      sx_ReqInProgress380 { ExternalAccessible := 'False'; ExternalVisible := 'False'; ExternalWritable := 'False'} : Bool;   // Request for 380 is in progress
      sx_ReqInProgress390 { ExternalAccessible := 'False'; ExternalVisible := 'False'; ExternalWritable := 'False'} : Bool;   // Request for 390 is in progress
      sx_ActiveRequest680 { ExternalAccessible := 'False'; ExternalVisible := 'False'; ExternalWritable := 'False'} : Bool;   // Request for 680 is active
      sx_ActiveRequest690 { ExternalAccessible := 'False'; ExternalVisible := 'False'; ExternalWritable := 'False'} : Bool;   // Request for 690 is active
      sx_ReqInProgress680 { ExternalAccessible := 'False'; ExternalVisible := 'False'; ExternalWritable := 'False'} : Bool;   // Request for 680 is in progress
      sx_ReqInProgress690 { ExternalAccessible := 'False'; ExternalVisible := 'False'; ExternalWritable := 'False'} : Bool;   // Request for 690 is in progress
      sx_TransferOut380 { ExternalAccessible := 'False'; ExternalVisible := 'False'; ExternalWritable := 'False'} : Bool;   // Transfer out from 380 is active
      sx_TransferOut390 { ExternalAccessible := 'False'; ExternalVisible := 'False'; ExternalWritable := 'False'} : Bool;   // Transfer out from 390 is active
      sx_TransferOut680 { ExternalAccessible := 'False'; ExternalVisible := 'False'; ExternalWritable := 'False'} : Bool;   // Transfer out from 680 is active
      sx_TransferOut690 { ExternalAccessible := 'False'; ExternalVisible := 'False'; ExternalWritable := 'False'} : Bool;   // Transfer out from 690 is active
      sx_DirectionChange380 { ExternalAccessible := 'False'; ExternalVisible := 'False'; ExternalWritable := 'False'} : Bool;   // Direction of conveyor 380
      sx_DirectionChange390 { ExternalAccessible := 'False'; ExternalVisible := 'False'; ExternalWritable := 'False'} : Bool;   // Direction of conveyor 390
      sx_DirectionChange680 { ExternalAccessible := 'False'; ExternalVisible := 'False'; ExternalWritable := 'False'} : Bool;   // Direction of conveyor 680
      sx_DirectionChange690 { ExternalAccessible := 'False'; ExternalVisible := 'False'; ExternalWritable := 'False'} : Bool;   // Direction of conveyor 690
      sx_Hold230 { ExternalAccessible := 'False'; ExternalVisible := 'False'; ExternalWritable := 'False'} : Bool;
      sx_Hold530 { ExternalAccessible := 'False'; ExternalVisible := 'False'; ExternalWritable := 'False'} : Bool;
      sx_ClearRightStation { ExternalAccessible := 'False'; ExternalVisible := 'False'; ExternalWritable := 'False'} : Bool;   // Command to clear right station
      sx_ClearLeftStation { ExternalAccessible := 'False'; ExternalVisible := 'False'; ExternalWritable := 'False'} : Bool;   // Command to clear left station
   END_VAR

   VAR_TEMP
      tUDT_dummyHandshake : "UDT_ConveyorHandshake";   // Dummy handshake structure
      tUDT_DummyBladeStop : "UDT_ValveInterface";
      ts_Barcode110 : String;
      ts_Barcode330 : String;
      ts_Barcode630 : String;
      tw_dummy : Word;
      ti_dummy : Int;   // Dummy int
      tx_dummy : Bool;   // Dummy bool
   END_VAR


BEGIN
	(*
	----------------------------------------------------------------------------------------

	Version history:
	Date        | Version   | Author        | Remark
	----------------------------------------------------------------------------------------
	23/02/2024  | 0.1       | R. Pieczonka  | Initial version
	26/02/2024  | 0.2       | S. Nieswiec   | Updated to new library blocks, added HardwareOk input
	27/02/2024  | 0.3       | S. Nieswiec   | Mapped  safetyOk, 24vOk, 400vOk from inputs to function blocks, added VFDs in place of conveylinx at conveyors 260,310,560,610
	18/03/2024  | 0.4       | S. Nieswiec   | Adjusted comments and variable names
	15/04/2024  | 0.5       | S. Nieswiec   | Added ConveyLinx Controllers
	10/05/2024  | 0.6       | R. Pieczonka  | Added new MCO and clearing sequence. Changes in station operation sequence.
	04/06/2024  | 0.7       | S. Nieswiec   | Partially added scanners
	11/06/2024  | 0.8       | S. Nieswiec   | New RAT, MCO and Displacement FB + added datalogic scanner
	14/06/2024  | 0.9       | S. Nieswiec   | New RAT, MCO and Displacement FB + added datalogic scanner
	*)
	(*
	----------------------------------------------------------------------------------------

	Notes:
	Date        | Version   | Author        | Notes
	----------------------------------------------------------------------------------------
	25/06/2024  | 0.9       | I.Bou Ajram   | Barcode scanners and the use of external DBs directly needs tidying up. request update


	*)

	REGION Middle line - Infeed
	    (*
	    REGION 010

	        REGION Displacement

	            #sFB_Displacement010(#sUDT_Interface_010);

	        END_REGION

	        REGION Conveyor
	            #sFB_Conveyor_010(iUDT_ConveyorConfiguration := #iUDT_Configuration."010".Conveyor,
	                              idi_PECEoSDistance         := 0,
	                              idi_PECBoSDistance         := 0,
	                              ii_ExternalSpeed           := 0,
	                              ix_SafetyOk                := #ix_SafetyOk,
	                              ix_24vOk                   := #ix_24vOk,
	                              ix_400vOk                  := #ix_400vOk,
	                              ix_HardwareOk              := #ix_HardwareOk,
	                              ix_PECEoS                  := TRUE,
	                              ix_PECBoS                  := TRUE,
	                              ix_ExternalRequestHold     := false,
	                              qUDT_HMIStatus             => #iqUDT_WorkstationStatus."010".Conveyor,
	                              qUDT_Status                => #iqUDT_WorkstationCommonStatus."010",
	                              iqUDT_EquipmentControl     := #iqUDT_EquipmentControl,
	                              iqUDT_ConveyorCommand      := #iqUDT_WorkstationCommands."010",
	                              iqUDT_ConveyorInterface    := #sUDT_Interface_010,
	                              iqUDT_HandShakeUp          := #iqUDT_HandshakeUpstream010,
	                              iqUDT_HandShake            := #sUDT_Handshake_010,
	                              iqUDT_Statistics           := #iqUDT_WorkstationStatistics."010".Conveyor);
	        END_REGION

	        REGION MCO
	            #sFB_MCOConveyLinxAixController_010(iUDT_AixConfig          := #iUDT_Configuration."010".MCO,
	                                                iUDT_AixInputsModule    := #iUDT_MotorInput010,
	                                                ix_24vOk                := #ix_24vOk,
	                                                ix_SimulationModeActive := "DB_Memory".Simulation,
	                                                ii_MotorPositionId      := 1,
	                                                qUDT_HMIStatus          => #iqUDT_WorkstationStatus."010".MCO,
	                                                iqUDT_AixOutputsModule  := #qUDT_MotorOutput010,
	                                                iqUDT_ConveyorInterface := #sUDT_Interface_010,
	                                                iqUDT_MCOStatistics     := #iqUDT_WorkstationStatistics."010".MCO);
	        END_REGION
	    END_REGION


	    REGION 020

	        REGION Displacement

	            #sFB_Displacement020(#sUDT_Interface_020);

	        END_REGION

	        REGION EoS

	            #sFB_PEC_020(ix_PEC                   := #iUDT_MotorInput020.AllSensorPortInputs.LeftSensor,
	                         iUDT_PECConfiguration   := #iUDT_Configuration."020".PEC_Eos,
	                         qUDT_HMIStatus          => #iqUDT_WorkstationStatus."020".PEC_Eos,
	                         iqUDT_ConveyorInterface := #sUDT_Interface_020,
	                         iqUDT_PECStatistics     := #iqUDT_WorkstationStatistics."020".PEC_Eos);

	        END_REGION

	        REGION Conveyor
	            #sFB_Conveyor_020(iUDT_ConveyorConfiguration := #iUDT_Configuration."020".Conveyor,
	                              idi_PECEoSDistance         := #iUDT_Configuration."020".PEC_Eos.Distance,
	                              idi_PECBoSDistance         := 0,
	                              ii_ExternalSpeed           := 0,
	                              ix_SafetyOk                := #ix_SafetyOk,
	                              ix_24vOk                   := #ix_24vOk,
	                              ix_400vOk                  := #ix_400vOk,
	                              ix_HardwareOk              := #ix_HardwareOk,
	                              ix_PECEoS                  := #iqUDT_WorkstationStatus."020".PEC_Eos.PEC,
	                              ix_PECBoS                  := TRUE,
	                              ix_ExternalRequestHold     := false,
	                              qUDT_HMIStatus             => #iqUDT_WorkstationStatus."020".Conveyor,
	                              qUDT_Status                => #iqUDT_WorkstationCommonStatus."020",
	                              iqUDT_EquipmentControl     := #iqUDT_EquipmentControl,
	                              iqUDT_ConveyorCommand      := #iqUDT_WorkstationCommands."020",
	                              iqUDT_ConveyorInterface    := #sUDT_Interface_020,
	                              iqUDT_HandShakeUp          := #sUDT_Handshake_010,
	                              iqUDT_HandShake            := #sUDT_Handshake_020,
	                              iqUDT_Statistics           := #iqUDT_WorkstationStatistics."020".Conveyor);
	        END_REGION

	        REGION MCO
	            #sFB_MCOConveyLinxAixController_020(iUDT_AixConfig          := #iUDT_Configuration."020".MCO,
	                                                iUDT_AixInputsModule    := #iUDT_MotorInput020,
	                                                ix_24vOk                := #ix_24vOk,
	                                                ix_SimulationModeActive := "DB_Memory".Simulation,
	                                                ii_MotorPositionId      := 1,
	                                                qUDT_HMIStatus          => #iqUDT_WorkstationStatus."020".MCO,
	                                                iqUDT_AixOutputsModule  := #qUDT_MotorOutput020,
	                                                iqUDT_ConveyorInterface := #sUDT_Interface_020,
	                                                iqUDT_MCOStatistics     := #iqUDT_WorkstationStatistics."020".MCO);
	        END_REGION


	    END_REGION

	    REGION 030

	        REGION Displacement

	            #sFB_Displacement030(#sUDT_Interface_030);

	        END_REGION

	        REGION EoS

	            #sFB_PEC_030(ix_PEC                   := #iUDT_MotorInput030.AllSensorPortInputs.LeftSensor,
	                         iUDT_PECConfiguration   := #iUDT_Configuration."030".PEC_Eos,
	                         qUDT_HMIStatus          => #iqUDT_WorkstationStatus."030".PEC_Eos,
	                         iqUDT_ConveyorInterface := #sUDT_Interface_030,
	                         iqUDT_PECStatistics     := #iqUDT_WorkstationStatistics."030".PEC_Eos);

	        END_REGION

	        REGION Conveyor
	            #sFB_Conveyor_030(iUDT_ConveyorConfiguration := #iUDT_Configuration."030".Conveyor,
	                              idi_PECEoSDistance         := #iUDT_Configuration."030".PEC_Eos.Distance,
	                              idi_PECBoSDistance         := 0,
	                              ii_ExternalSpeed           := 0,
	                              ix_SafetyOk                := #ix_SafetyOk,
	                              ix_24vOk                   := #ix_24vOk,
	                              ix_400vOk                  := #ix_400vOk,
	                              ix_HardwareOk              := #ix_HardwareOk,
	                              ix_PECEoS                  := #iqUDT_WorkstationStatus."030".PEC_Eos.PEC,
	                              ix_PECBoS                  := TRUE,
	                              ix_ExternalRequestHold     := false,
	                              qUDT_HMIStatus             => #iqUDT_WorkstationStatus."030".Conveyor,
	                              qUDT_Status                => #iqUDT_WorkstationCommonStatus."030",
	                              iqUDT_EquipmentControl     := #iqUDT_EquipmentControl,
	                              iqUDT_ConveyorCommand      := #iqUDT_WorkstationCommands."030",
	                              iqUDT_ConveyorInterface    := #sUDT_Interface_030,
	                              iqUDT_HandShakeUp          := #sUDT_Handshake_020,
	                              iqUDT_HandShake            := #sUDT_Handshake_030,
	                              iqUDT_Statistics           := #iqUDT_WorkstationStatistics."030".Conveyor);
	        END_REGION

	        REGION MCO
	            #sFB_MCOConveyLinxAixController_030(iUDT_AixConfig          := #iUDT_Configuration."030".MCO,
	                                                iUDT_AixInputsModule    := #iUDT_MotorInput030,
	                                                ix_24vOk                := #ix_24vOk,
	                                                ix_SimulationModeActive := "DB_Memory".Simulation,
	                                                ii_MotorPositionId      := 1,
	                                                qUDT_HMIStatus          => #iqUDT_WorkstationStatus."030".MCO,
	                                                iqUDT_AixOutputsModule  := #qUDT_MotorOutput030,
	                                                iqUDT_ConveyorInterface := #sUDT_Interface_030,
	                                                iqUDT_MCOStatistics     := #iqUDT_WorkstationStatistics."030".MCO);
	        END_REGION
	    END_REGION

	    REGION 040

	        REGION Displacement

	            #sFB_Displacement040(#sUDT_Interface_040);

	        END_REGION

	        REGION EoS

	            #sFB_PEC_040(ix_PEC                   := #iUDT_MotorInput040.AllSensorPortInputs.LeftSensor,
	                         iUDT_PECConfiguration   := #iUDT_Configuration."040".PEC_Eos,
	                         qUDT_HMIStatus          => #iqUDT_WorkstationStatus."040".PEC_Eos,
	                         iqUDT_ConveyorInterface := #sUDT_Interface_040,
	                         iqUDT_PECStatistics     := #iqUDT_WorkstationStatistics."040".PEC_Eos);

	        END_REGION

	        REGION Conveyor
	            #sFB_Conveyor_040(iUDT_ConveyorConfiguration := #iUDT_Configuration."040".Conveyor,
	                              idi_PECEoSDistance         := #iUDT_Configuration."040".PEC_Eos.Distance,
	                              idi_PECBoSDistance         := 0,
	                              ii_ExternalSpeed           := 0,
	                              ix_SafetyOk                := #ix_SafetyOk,
	                              ix_24vOk                   := #ix_24vOk,
	                              ix_400vOk                  := #ix_400vOk,
	                              ix_HardwareOk              := #ix_HardwareOk,
	                              ix_PECEoS                  := #iqUDT_WorkstationStatus."040".PEC_Eos.PEC,
	                              ix_PECBoS                  := TRUE,
	                              ix_ExternalRequestHold     := false,
	                              qUDT_HMIStatus             => #iqUDT_WorkstationStatus."040".Conveyor,
	                              qUDT_Status                => #iqUDT_WorkstationCommonStatus."040",
	                              iqUDT_EquipmentControl     := #iqUDT_EquipmentControl,
	                              iqUDT_ConveyorCommand      := #iqUDT_WorkstationCommands."040",
	                              iqUDT_ConveyorInterface    := #sUDT_Interface_040,
	                              iqUDT_HandShakeUp          := #sUDT_Handshake_030,
	                              iqUDT_HandShake            := #sUDT_Handshake_040,
	                              iqUDT_Statistics           := #iqUDT_WorkstationStatistics."040".Conveyor);
	        END_REGION

	        REGION MCO
	            #sFB_MCOConveyLinxAixController_040(iUDT_AixConfig          := #iUDT_Configuration."040".MCO,
	                                                iUDT_AixInputsModule    := #iUDT_MotorInput040,
	                                                ix_24vOk                := #ix_24vOk,
	                                                ix_SimulationModeActive := "DB_Memory".Simulation,
	                                                ii_MotorPositionId      := 1,
	                                                qUDT_HMIStatus          => #iqUDT_WorkstationStatus."040".MCO,
	                                                iqUDT_AixOutputsModule  := #qUDT_MotorOutput040,
	                                                iqUDT_ConveyorInterface := #sUDT_Interface_040,
	                                                iqUDT_MCOStatistics     := #iqUDT_WorkstationStatistics."040".MCO);
	        END_REGION

	    END_REGION

	    REGION 050

	        REGION Displacement

	            #sFB_Displacement050(#sUDT_Interface_050);

	        END_REGION

	        REGION EoS

	            #sFB_PEC_050(ix_PEC                   := #iUDT_MotorInput050.AllSensorPortInputs.LeftSensor,
	                         iUDT_PECConfiguration   := #iUDT_Configuration."050".PEC_Eos,
	                         qUDT_HMIStatus          => #iqUDT_WorkstationStatus."050".PEC_Eos,
	                         iqUDT_ConveyorInterface := #sUDT_Interface_050,
	                         iqUDT_PECStatistics     := #iqUDT_WorkstationStatistics."050".PEC_Eos);

	        END_REGION

	        REGION Conveyor
	            #sFB_Conveyor_050(iUDT_ConveyorConfiguration := #iUDT_Configuration."050".Conveyor,
	                              idi_PECEoSDistance         := #iUDT_Configuration."050".PEC_Eos.Distance,
	                              idi_PECBoSDistance         := 0,
	                              ii_ExternalSpeed           := 0,
	                              ix_SafetyOk                := #ix_SafetyOk,
	                              ix_24vOk                   := #ix_24vOk,
	                              ix_400vOk                  := #ix_400vOk,
	                              ix_HardwareOk              := #ix_HardwareOk,
	                              ix_PECEoS                  := #iqUDT_WorkstationStatus."050".PEC_Eos.PEC,
	                              ix_PECBoS                  := TRUE,
	                              ix_ExternalRequestHold     := false,
	                              qUDT_HMIStatus             => #iqUDT_WorkstationStatus."050".Conveyor,
	                              qUDT_Status                => #iqUDT_WorkstationCommonStatus."050",
	                              iqUDT_EquipmentControl     := #iqUDT_EquipmentControl,
	                              iqUDT_ConveyorCommand      := #iqUDT_WorkstationCommands."050",
	                              iqUDT_ConveyorInterface    := #sUDT_Interface_050,
	                              iqUDT_HandShakeUp          := #sUDT_Handshake_040,
	                              iqUDT_HandShake            := #sUDT_Handshake_050,
	                              iqUDT_Statistics           := #iqUDT_WorkstationStatistics."050".Conveyor);
	        END_REGION

	        REGION MCO
	            #sFB_MCOConveyLinxAixController_050(iUDT_AixConfig          := #iUDT_Configuration."050".MCO,
	                                                iUDT_AixInputsModule    := #iUDT_MotorInput050,
	                                                ix_24vOk                := #ix_24vOk,
	                                                ix_SimulationModeActive := "DB_Memory".Simulation,
	                                                ii_MotorPositionId      := 1,
	                                                qUDT_HMIStatus          => #iqUDT_WorkstationStatus."050".MCO,
	                                                iqUDT_AixOutputsModule  := #qUDT_MotorOutput050,
	                                                iqUDT_ConveyorInterface := #sUDT_Interface_050,
	                                                iqUDT_MCOStatistics     := #iqUDT_WorkstationStatistics."050".MCO);
	        END_REGION
	    END_REGION

	    REGION 060

	        REGION Displacement

	            #sFB_Displacement060(#sUDT_Interface_060);

	        END_REGION

	        REGION EoS

	            #sFB_PEC_060(ix_PEC                   := #iUDT_MotorInput060.AllSensorPortInputs.LeftSensor,
	                         iUDT_PECConfiguration   := #iUDT_Configuration."060".PEC_Eos,
	                         qUDT_HMIStatus          => #iqUDT_WorkstationStatus."060".PEC_Eos,
	                         iqUDT_ConveyorInterface := #sUDT_Interface_060,
	                         iqUDT_PECStatistics     := #iqUDT_WorkstationStatistics."060".PEC_Eos);

	        END_REGION

	        REGION Conveyor
	            #sFB_Conveyor_060(iUDT_ConveyorConfiguration := #iUDT_Configuration."060".Conveyor,
	                              idi_PECEoSDistance         := #iUDT_Configuration."060".PEC_Eos.Distance,
	                              idi_PECBoSDistance         := 0,
	                              ii_ExternalSpeed           := 0,
	                              ix_SafetyOk                := #ix_SafetyOk,
	                              ix_24vOk                   := #ix_24vOk,
	                              ix_400vOk                  := #ix_400vOk,
	                              ix_HardwareOk              := #ix_HardwareOk,
	                              ix_PECEoS                  := #iqUDT_WorkstationStatus."060".PEC_Eos.PEC,
	                              ix_PECBoS                  := TRUE,
	                              ix_ExternalRequestHold     := false,
	                              qUDT_HMIStatus             => #iqUDT_WorkstationStatus."060".Conveyor,
	                              qUDT_Status                => #iqUDT_WorkstationCommonStatus."060",
	                              iqUDT_EquipmentControl     := #iqUDT_EquipmentControl,
	                              iqUDT_ConveyorCommand      := #iqUDT_WorkstationCommands."060",
	                              iqUDT_ConveyorInterface    := #sUDT_Interface_060,
	                              iqUDT_HandShakeUp          := #sUDT_Handshake_050,
	                              iqUDT_HandShake            := #sUDT_Handshake_060,
	                              iqUDT_Statistics           := #iqUDT_WorkstationStatistics."060".Conveyor);
	        END_REGION

	        REGION MCO
	            #sFB_MCOConveyLinxAixController_060(iUDT_AixConfig          := #iUDT_Configuration."060".MCO,
	                                                iUDT_AixInputsModule    := #iUDT_MotorInput060,
	                                                ix_24vOk                := #ix_24vOk,
	                                                ix_SimulationModeActive := "DB_Memory".Simulation,
	                                                ii_MotorPositionId      := 1,
	                                                qUDT_HMIStatus          => #iqUDT_WorkstationStatus."060".MCO,
	                                                iqUDT_AixOutputsModule  := #qUDT_MotorOutput060,
	                                                iqUDT_ConveyorInterface := #sUDT_Interface_060,
	                                                iqUDT_MCOStatistics     := #iqUDT_WorkstationStatistics."060".MCO);
	        END_REGION

	    END_REGION

	    REGION 070

	        REGION Displacement

	            #sFB_Displacement070(#sUDT_Interface_070);

	        END_REGION

	        REGION EoS

	            #sFB_PEC_070(ix_PEC                   := #iUDT_MotorInput070.AllSensorPortInputs.LeftSensor,
	                         iUDT_PECConfiguration   := #iUDT_Configuration."070".PEC_Eos,
	                         qUDT_HMIStatus          => #iqUDT_WorkstationStatus."070".PEC_Eos,
	                         iqUDT_ConveyorInterface := #sUDT_Interface_070,
	                         iqUDT_PECStatistics     := #iqUDT_WorkstationStatistics."070".PEC_Eos);

	        END_REGION

	        REGION Conveyor
	            #sFB_Conveyor_070(iUDT_ConveyorConfiguration := #iUDT_Configuration."070".Conveyor,
	                              idi_PECEoSDistance         := #iUDT_Configuration."070".PEC_Eos.Distance,
	                              idi_PECBoSDistance         := 0,
	                              ii_ExternalSpeed           := 0,
	                              ix_SafetyOk                := #ix_SafetyOk,
	                              ix_24vOk                   := #ix_24vOk,
	                              ix_400vOk                  := #ix_400vOk,
	                              ix_HardwareOk              := #ix_HardwareOk,
	                              ix_PECEoS                  := #iqUDT_WorkstationStatus."070".PEC_Eos.PEC,
	                              ix_PECBoS                  := TRUE,
	                              ix_ExternalRequestHold     := false,
	                              qUDT_HMIStatus             => #iqUDT_WorkstationStatus."070".Conveyor,
	                              qUDT_Status                => #iqUDT_WorkstationCommonStatus."070",
	                              iqUDT_EquipmentControl     := #iqUDT_EquipmentControl,
	                              iqUDT_ConveyorCommand      := #iqUDT_WorkstationCommands."070",
	                              iqUDT_ConveyorInterface    := #sUDT_Interface_070,
	                              iqUDT_HandShakeUp          := #sUDT_Handshake_060,
	                              iqUDT_HandShake            := #sUDT_Handshake_070,
	                              iqUDT_Statistics           := #iqUDT_WorkstationStatistics."070".Conveyor);
	        END_REGION

	        REGION MCO
	            #sFB_MCOConveyLinxAixController_070(iUDT_AixConfig          := #iUDT_Configuration."070".MCO,
	                                                iUDT_AixInputsModule    := #iUDT_MotorInput070,
	                                                ix_24vOk                := #ix_24vOk,
	                                                ix_SimulationModeActive := "DB_Memory".Simulation,
	                                                ii_MotorPositionId      := 1,
	                                                qUDT_HMIStatus          => #iqUDT_WorkstationStatus."070".MCO,
	                                                iqUDT_AixOutputsModule  := #qUDT_MotorOutput070,
	                                                iqUDT_ConveyorInterface := #sUDT_Interface_070,
	                                                iqUDT_MCOStatistics     := #iqUDT_WorkstationStatistics."070".MCO);
	        END_REGION
	    END_REGION

	    REGION 080

	        REGION Displacement

	            #sFB_Displacement080(#sUDT_Interface_080);

	        END_REGION

	        REGION EoS

	            #sFB_PEC_080(ix_PEC                   := #iUDT_MotorInput080.AllSensorPortInputs.LeftSensor,
	                         iUDT_PECConfiguration   := #iUDT_Configuration."080".PEC_Eos,
	                         qUDT_HMIStatus          => #iqUDT_WorkstationStatus."080".PEC_Eos,
	                         iqUDT_ConveyorInterface := #sUDT_Interface_080,
	                         iqUDT_PECStatistics     := #iqUDT_WorkstationStatistics."080".PEC_Eos);

	        END_REGION

	        REGION Conveyor
	            #sFB_Conveyor_080(iUDT_ConveyorConfiguration := #iUDT_Configuration."080".Conveyor,
	                              idi_PECEoSDistance         := #iUDT_Configuration."080".PEC_Eos.Distance,
	                              idi_PECBoSDistance         := 0,
	                              ii_ExternalSpeed           := 0,
	                              ix_SafetyOk                := #ix_SafetyOk,
	                              ix_24vOk                   := #ix_24vOk,
	                              ix_400vOk                  := #ix_400vOk,
	                              ix_HardwareOk              := #ix_HardwareOk,
	                              ix_PECEoS                  := #iqUDT_WorkstationStatus."080".PEC_Eos.PEC,
	                              ix_PECBoS                  := TRUE,
	                              ix_ExternalRequestHold     := false,
	                              qUDT_HMIStatus             => #iqUDT_WorkstationStatus."080".Conveyor,
	                              qUDT_Status                => #iqUDT_WorkstationCommonStatus."080",
	                              iqUDT_EquipmentControl     := #iqUDT_EquipmentControl,
	                              iqUDT_ConveyorCommand      := #iqUDT_WorkstationCommands."080",
	                              iqUDT_ConveyorInterface    := #sUDT_Interface_080,
	                              iqUDT_HandShakeUp          := #sUDT_Handshake_070,
	                              iqUDT_HandShake            := #sUDT_Handshake_080,
	                              iqUDT_Statistics           := #iqUDT_WorkstationStatistics."080".Conveyor);
	        END_REGION

	        REGION MCO
	            #sFB_MCOConveyLinxAixController_080(iUDT_AixConfig          := #iUDT_Configuration."080".MCO,
	                                                iUDT_AixInputsModule    := #iUDT_MotorInput080,
	                                                ix_24vOk                := #ix_24vOk,
	                                                ix_SimulationModeActive := "DB_Memory".Simulation,
	                                                ii_MotorPositionId      := 1,
	                                                qUDT_HMIStatus          => #iqUDT_WorkstationStatus."080".MCO,
	                                                iqUDT_AixOutputsModule  := #qUDT_MotorOutput080,
	                                                iqUDT_ConveyorInterface := #sUDT_Interface_080,
	                                                iqUDT_MCOStatistics     := #iqUDT_WorkstationStatistics."080".MCO);
	        END_REGION
	    END_REGION

	    REGION 090

	        REGION Displacement

	            #sFB_Displacement090(#sUDT_Interface_090);

	        END_REGION

	        REGION Conveyor
	            #sFB_Conveyor_090(iUDT_ConveyorConfiguration := #iUDT_Configuration."090".Conveyor,
	                              idi_PECEoSDistance         := 0,
	                              idi_PECBoSDistance         := 0,
	                              ii_ExternalSpeed           := 0,
	                              ix_SafetyOk                := #ix_SafetyOk,
	                              ix_24vOk                   := #ix_24vOk,
	                              ix_400vOk                  := #ix_400vOk,
	                              ix_HardwareOk              := #ix_HardwareOk,
	                              ix_PECEoS                  := TRUE,
	                              ix_PECBoS                  := TRUE,
	                              ix_ExternalRequestHold     := false,
	                              qUDT_HMIStatus             => #iqUDT_WorkstationStatus."090".Conveyor,
	                              qUDT_Status                => #iqUDT_WorkstationCommonStatus."090",
	                              iqUDT_EquipmentControl     := #iqUDT_EquipmentControl,
	                              iqUDT_ConveyorCommand      := #iqUDT_WorkstationCommands."090",
	                              iqUDT_ConveyorInterface    := #sUDT_Interface_090,
	                              iqUDT_HandShakeUp          := #sUDT_Handshake_080,
	                              iqUDT_HandShake            := #sUDT_Handshake_090,
	                              iqUDT_Statistics           := #iqUDT_WorkstationStatistics."090".Conveyor);
	        END_REGION

	        REGION MCO
	            #sFB_MCOConveyLinxAixController_090(iUDT_AixConfig          := #iUDT_Configuration."090".MCO,
	                                                iUDT_AixInputsModule    := #iUDT_MotorInput090,
	                                                ix_24vOk                := #ix_24vOk,
	                                                ix_SimulationModeActive := "DB_Memory".Simulation,
	                                                ii_MotorPositionId      := 1,
	                                                qUDT_HMIStatus          => #iqUDT_WorkstationStatus."090".MCO,
	                                                iqUDT_AixOutputsModule  := #qUDT_MotorOutput090,
	                                                iqUDT_ConveyorInterface := #sUDT_Interface_090,
	                                                iqUDT_MCOStatistics     := #iqUDT_WorkstationStatistics."090".MCO);
	        END_REGION
	    END_REGION

	    REGION 100

	        REGION Displacement

	            #sFB_Displacement100(#sUDT_Interface_100);

	        END_REGION

	        REGION EoS

	            #sFB_PEC_100(ix_PEC                   := #iUDT_MotorInput100.AllSensorPortInputs.LeftSensor,
	                         iUDT_PECConfiguration   := #iUDT_Configuration."100".PEC_Eos,
	                         qUDT_HMIStatus          => #iqUDT_WorkstationStatus."100".PEC_Eos,
	                         iqUDT_ConveyorInterface := #sUDT_Interface_100,
	                         iqUDT_PECStatistics     := #iqUDT_WorkstationStatistics."100".PEC_Eos);

	        END_REGION

	        REGION Conveyor
	            #sFB_Conveyor_100(iUDT_ConveyorConfiguration := #iUDT_Configuration."100".Conveyor,
	                              idi_PECEoSDistance         := #iUDT_Configuration."100".PEC_Eos.Distance,
	                              idi_PECBoSDistance         := 0,
	                              ii_ExternalSpeed           := 0,
	                              ix_SafetyOk                := #ix_SafetyOk,
	                              ix_24vOk                   := #ix_24vOk,
	                              ix_400vOk                  := #ix_400vOk,
	                              ix_HardwareOk              := #ix_HardwareOk,
	                              ix_PECEoS                  := #iqUDT_WorkstationStatus."100".PEC_Eos.PEC,
	                              ix_PECBoS                  := TRUE,
	                              ix_ExternalRequestHold     := false,
	                              qUDT_HMIStatus             => #iqUDT_WorkstationStatus."100".Conveyor,
	                              qUDT_Status                => #iqUDT_WorkstationCommonStatus."100",
	                              iqUDT_EquipmentControl     := #iqUDT_EquipmentControl,
	                              iqUDT_ConveyorCommand      := #iqUDT_WorkstationCommands."100",
	                              iqUDT_ConveyorInterface    := #sUDT_Interface_100,
	                              iqUDT_HandShakeUp          := #sUDT_Handshake_090,
	                              iqUDT_HandShake            := #sUDT_Handshake_100,
	                              iqUDT_Statistics           := #iqUDT_WorkstationStatistics."100".Conveyor);
	        END_REGION

	        REGION MCO
	            #sFB_MCOConveyLinxAixController_100(iUDT_AixConfig          := #iUDT_Configuration."100".MCO,
	                                                iUDT_AixInputsModule    := #iUDT_MotorInput100,
	                                                ix_24vOk                := #ix_24vOk,
	                                                ix_SimulationModeActive := "DB_Memory".Simulation,
	                                                ii_MotorPositionId      := 1,
	                                                qUDT_HMIStatus          => #iqUDT_WorkstationStatus."100".MCO,
	                                                iqUDT_AixOutputsModule  := #qUDT_MotorOutput100,
	                                                iqUDT_ConveyorInterface := #sUDT_Interface_100,
	                                                iqUDT_MCOStatistics     := #iqUDT_WorkstationStatistics."100".MCO);
	        END_REGION

	    END_REGION

	    REGION 110

	        REGION Displacement

	            #sFB_Displacement110(#sUDT_Interface_110);

	        END_REGION

	        REGION EoS

	            #sFB_PEC_110(ix_PEC                   := #iUDT_MotorInput110.AllSensorPortInputs.LeftSensor,
	                         iUDT_PECConfiguration   := #iUDT_Configuration."110".PEC_Eos,
	                         qUDT_HMIStatus          => #iqUDT_WorkstationStatus."110".PEC_Eos,
	                         iqUDT_ConveyorInterface := #sUDT_Interface_110,
	                         iqUDT_PECStatistics     := #iqUDT_WorkstationStatistics."110".PEC_Eos);

	        END_REGION

	        REGION Scanner

	            #sFB_CognexDM260_110(iUDT_CognexDM260_IN    := #iUDT_ScannerInput110,
	                                 qs_Barcode             => #ts_Barcode110,
	                                 iqUDT_EquipmentControl := #iqUDT_EquipmentControl,
	                                 ix_Trigger             := #tx_dummy,
	                                 qUDT_CognexDM260_OUT   => #qUDT_ScannerOutput110,
	                                 qw_RetVal              => #tw_dummy);

	        END_REGION

	        REGION Conveyor
	            #sUDT_Handshake_110.RTR := #sUDT_Handshake_110.RTR OR #iqUDT_WorkstationStatus."110".PEC_Eos.PEC;
	            #sFB_Conveyor_110(iUDT_ConveyorConfiguration := #iUDT_Configuration."110".Conveyor,
	                              idi_PECEoSDistance         := #iUDT_Configuration."110".PEC_Eos.Distance,
	                              idi_PECBoSDistance         := 0,
	                              ii_ExternalSpeed           := 0,
	                              ix_SafetyOk                := #ix_SafetyOk,
	                              ix_24vOk                   := #ix_24vOk,
	                              ix_400vOk                  := #ix_400vOk,
	                              ix_HardwareOk              := #ix_HardwareOk,
	                              ix_PECEoS                  := #iqUDT_WorkstationStatus."110".PEC_Eos.PEC,
	                              ix_PECBoS                  := TRUE,
	                              ix_ExternalRequestHold     := false,
	                              qUDT_HMIStatus             => #iqUDT_WorkstationStatus."110".Conveyor,
	                              qUDT_Status                => #iqUDT_WorkstationCommonStatus."110",
	                              iqUDT_EquipmentControl     := #iqUDT_EquipmentControl,
	                              iqUDT_ConveyorCommand      := #iqUDT_WorkstationCommands."110",
	                              iqUDT_ConveyorInterface    := #sUDT_Interface_110,
	                              iqUDT_HandShakeUp          := #sUDT_Handshake_100,
	                              iqUDT_HandShake            := #sUDT_Handshake_110,
	                              iqUDT_Statistics           := #iqUDT_WorkstationStatistics."110".Conveyor);
	        END_REGION

	        REGION MCO
	            #sFB_MCOConveyLinxAixController_110(iUDT_AixConfig          := #iUDT_Configuration."110".MCO,
	                                                iUDT_AixInputsModule    := #iUDT_MotorInput110,
	                                                ix_24vOk                := #ix_24vOk,
	                                                ix_SimulationModeActive := "DB_Memory".Simulation,
	                                                ii_MotorPositionId      := 1,
	                                                qUDT_HMIStatus          => #iqUDT_WorkstationStatus."110".MCO,
	                                                iqUDT_AixOutputsModule  := #qUDT_MotorOutput110,
	                                                iqUDT_ConveyorInterface := #sUDT_Interface_110,
	                                                iqUDT_MCOStatistics     := #iqUDT_WorkstationStatistics."110".MCO);
	        END_REGION
	    END_REGION

	    REGION 120

	        REGION Displacement

	            #sFB_Displacement120(#sUDT_Interface_120);

	        END_REGION

	        REGION MCO
	            #sFB_MCOConveyLinxAixController_120(iUDT_AixConfig          := #iUDT_Configuration."120".MCO,
	                                                iUDT_AixInputsModule    := #iUDT_MotorInput120,
	                                                ii_PositionSetpoint     := #iqUDT_RATPositioning120.Lower.EndPosition,
	                                                ix_24vOk                := #ix_24vOk,
	                                                ix_SimulationModeActive := "DB_Memory".Simulation,
	                                                ii_MotorPositionId      := 1,
	                                                ix_StartPositioning     := #iqUDT_RATPositioning120.Lower.Start,
	                                                ix_ResetPosition        := #iqUDT_RATPositioning120.Lower.ResetPosition,
	                                                qUDT_HMIStatus          => #iqUDT_WorkstationStatus."120".MCO,
	                                                qx_Positioned           => #iqUDT_RATPositioning120.Lower.Done,
	                                                iqUDT_AixOutputsModule  := #qUDT_MotorOutput120,
	                                                iqUDT_ConveyorInterface := #sUDT_Interface_120,
	                                                iqUDT_MCOStatistics     := #iqUDT_WorkstationStatistics."120".MCO);
	        END_REGION


	    END_REGION

	    REGION 121

	        REGION RAT
	            //Destination from 120
	            IF #ix_LeftReqFromMid THEN
	                #si_120DestinationA := 2;
	                #si_120DestinationB := 0;
	                #si_120DestinationC := 0;
	                #si_120DestinationD := 0;
	            ELSIF #ix_RightReqFromMid THEN
	                #si_120DestinationA := 1;
	                #si_120DestinationB := 0;
	                #si_120DestinationC := 0;
	                #si_120DestinationD := 0;
	            ELSE
	                #si_120DestinationA := 0;
	                #si_120DestinationB := 0;
	                #si_120DestinationC := 0;
	                #si_120DestinationD := 0;
	            END_IF;

	            #sUDT_HandshakeUp_121.RTR := TRUE;
	            #sUDT_Handshake_121.RTR := TRUE;

	    IF #sUDT_Interface_120.ActualSpeed = 0 AND NOT #iqUDT_WorkstationStatus."120".PEC_Eos.PEC THEN
	                "qx_WSV01-221-S11_Light" := TRUE;
	                "qx_WSV01-521-S11_Light" := TRUE;
	            ELSE
	                "qx_WSV01-221-S11_Light" := FALSE;
	                "qx_WSV01-521-S11_Light" := FALSE;
	            END_IF;

	            #sFB_RightAngledTransfer_121(iUDT_Configuration              := #iUDT_Configuration."121".RAT,
	                                         iUDT_LowerConveyorConfiguration := #iUDT_Configuration."120".Conveyor,
	                                         iUDT_UpperConveyorConfiguration := #iUDT_Configuration."121".Conveyor,
	                                         iUDT_PECConfiguration           := #iUDT_Configuration."120".PEC,
	                                         ii_DestinationA                 := #si_120DestinationA,
	                                         ii_DestinationB                 := #si_120DestinationB,
	                                         ii_DestinationC                 := #si_120DestinationC,
	                                         ii_DestinationD                 := #si_120DestinationD,
	                                         ix_HardwareOk                   := #ix_HardwareOk,
	                                         ix_400vOk                       := #ix_400vOk,
	                                         ix_24vOk                        := #ix_24vOk,
	                                         ix_SafetyOk                     := #ix_SafetyOk,
	                                         ix_AirPressureOk                := #ix_AirPressureOk,
	                                         ix_SectionIsDown                := #ix_SectionIsDown121,
	                                         ix_SectionIsUp                  := #ix_SectionIsUp121,
	                                         ix_ConveyorAAuto                := #iqUDT_WorkstationCommonStatus."110".AutoON,
	                                         ix_ConveyorBAuto                := false,
	                                         ix_ConveyorCAuto                := true,
	                                         ix_ConveyorDAuto                := true,
	                                         ix_PEC                          := #iUDT_MotorInput120.AllSensorPortInputs.LeftSensor,
	                                         ix_ExternalReceiveRequestA      := NOT #iqUDT_WorkstationStatus."110".PEC_Eos.PEC,
	                                         ix_ExternalReceiveRequestB      := false,
	                                         ix_ExternalReceiveRequestC      := false,
	                                         ix_ExternalReceiveRequestD      := false,
	                                         ix_PECInfeedA                   :=#iqUDT_WorkstationStatus."110".PEC_Eos.PEC,
	                                         qUDT_HMIRATStatus               => #iqUDT_WorkstationStatus."121".RAT,
	                                         qUDT_HMICovneyorStatus          => #iqUDT_WorkstationStatus."120".Conveyor,
	                                         qUDT_HMIPECStatus               => #iqUDT_WorkstationStatus."120".PEC_Eos,
	                                         qUDT_RATStatus                  => #iqUDT_WorkstationCommonStatus."121",
	                                         qUDT_ConveyorStatus             => #iqUDT_WorkstationCommonStatus."120",
	                                         qx_PopupControl                 => #qx_PopupControl121,
	                                         iqUDT_EquipmentControl          := #iqUDT_EquipmentControl,
	                                         iqUDT_RATCommand                := #iqUDT_WorkstationCommands."121",
	                                         iqUDT_ConveyorCommand           := #iqUDT_WorkstationCommands."120",
	                                         iqUDT_RATStatistics             := #iqUDT_WorkstationStatistics."121".RAT,
	                                         iqUDT_ConveyorStatistics        := #iqUDT_WorkstationStatistics."120".Conveyor,
	                                         iqUDT_PECStatistics             := #iqUDT_WorkstationStatistics."120".PEC_Eos,
	                                         iqUDT_HandShakeConveyorA        := #sUDT_Handshake_110,
	                                         iqUDT_HandShakeConveyorB        := #sUDT_Handshake_120,
	                                         iqUDT_HandShakeConveyorC        := #sUDT_HandshakeUp_121,
	                                         iqUDT_HandShakeConveyorD        := #sUDT_Handshake_121,
	                                         iqUDT_LowerConveyorInterface    := #sUDT_Interface_120,
	                                         iqUDT_UpperConveyorInterface    := #sUDT_Interface_121,
	                                         iqUDT_RATPositioning            := #iqUDT_RATPositioning120);

	        END_REGION
	        REGION MCO
	            #sFB_MCOConveyLinxAixController_121(iUDT_AixConfig          := #iUDT_Configuration."121".MCO,
	                                                iUDT_AixInputsModule    := #iUDT_MotorInput120,
	                                                ix_24vOk                := #ix_24vOk,
	                                                ix_SimulationModeActive := "DB_Memory".Simulation,
	                                                ii_MotorPositionId      := 2,
	                                                qUDT_HMIStatus          => #iqUDT_WorkstationStatus."121".MCO,
	                                                iqUDT_AixOutputsModule  := #qUDT_MotorOutput120,
	                                                iqUDT_ConveyorInterface := #sUDT_Interface_121,
	                                                iqUDT_MCOStatistics     := #iqUDT_WorkstationStatistics."121".MCO);
	        END_REGION
	    END_REGION*)
	END_REGION


	IF #iUDT_Configuration.GlobalConfig.RightStationExists THEN
	    REGION Right Station
	        REGION Right station control

	            //Triggers
	            #s_F_Trig_240(CLK := #iqUDT_WorkstationStatus."240".PEC_Eos.PEC);
	            #s_F_Trig_ClearRight(CLK := #sx_ClearRightStation);

	            //If any request comes, start if possible
	            IF #iqUDT_WorkstationStatus."380".PEC_Eos.PEC
	                AND #ix_StationActive
	                AND NOT #sx_ActiveRequest380
	                AND NOT #sx_TransferOut380
	                AND NOT #sx_ClearRightStation
	            THEN
	                #sx_ActiveRequest380 := TRUE;

	            END_IF;
	            IF #iqUDT_WorkstationStatus."390".PEC_Eos.PEC
	                AND #ix_StationActive
	                AND NOT #sx_ActiveRequest390
	                AND NOT #sx_TransferOut390
	                AND NOT #sx_ClearRightStation
	            THEN
	                #sx_ActiveRequest390 := TRUE;
	            END_IF;

	            //Request in progress
	            IF #sx_ActiveRequest380 AND #sFB_RightAngledTransfer_351.qx_ExternalSendRequestB
	            THEN
	                #sx_ReqInProgress380 := TRUE;
	            END_IF;

	            IF #sx_ActiveRequest390 AND #sFB_RightAngledTransfer_341.qx_ExternalSendRequestB
	            THEN
	                #sx_ReqInProgress390 := TRUE;
	            END_IF;

	            //Request fulfilled
	            IF #sx_ActiveRequest390 AND NOT #iqUDT_WorkstationStatus."390".PEC_Eos.PEC
	            THEN
	                #sx_ActiveRequest390 := FALSE;
	                #sx_ReqInProgress390 := FALSE;
	            END_IF;

	            IF #sx_ActiveRequest380 AND NOT #iqUDT_WorkstationStatus."390".PEC_Eos.PEC
	            THEN
	                #sx_ActiveRequest380 := FALSE;
	                #sx_ReqInProgress380 := FALSE;
	            END_IF;

	            //Start transfer out
	            IF #iqx_Done380
	                AND NOT #sx_TransferOut390
	                AND (#iqUDT_WorkstationStatus."240".PEC_Eos.PEC OR #sx_Hold230)
	                AND NOT #iqUDT_WorkstationStatus."380".PEC_Eos.PEC
	            THEN
	                #sx_TransferOut380 := TRUE;
	                #sx_Hold230 := TRUE;
	                #iqx_Done380 := FALSE;
	            END_IF;

	            IF #iqx_Done390
	                AND NOT #sx_TransferOut380
	                AND (#iqUDT_WorkstationStatus."240".PEC_Eos.PEC OR #sx_Hold230)
	                AND NOT #iqUDT_WorkstationStatus."390".PEC_Eos.PEC
	            THEN
	                #sx_TransferOut390 := TRUE;
	                #sx_Hold230 := TRUE;
	                #iqx_Done390 := FALSE;
	            END_IF;

	            //If transfer is in progress, set up directions and destinations
	            IF #sx_TransferOut380 THEN
	                #sx_DirectionChange380 := TRUE;
	            END_IF;

	            IF #sx_TransferOut390 THEN
	                #sx_DirectionChange390 := TRUE;
	            END_IF;

	            //If transfer is over set up directions and destinations

	            IF NOT #sx_TransferOut380 AND NOT #sx_TransferOut390 THEN
	                #sx_Hold230 := FALSE;
	            END_IF;

	            IF #sx_TransferOut380
	                AND #s_F_Trig_240.Q
	            THEN
	                #sx_TransferOut380 := FALSE;
	                #sx_DirectionChange380 := FALSE;
	            END_IF;

	            IF #sx_TransferOut390
	                AND #s_F_Trig_240.Q
	            THEN
	                #sx_TransferOut390 := FALSE;
	                #sx_DirectionChange390 := FALSE;
	            END_IF;


	            //Destinations from RAT 340
	            IF #sx_ActiveRequest390 AND NOT #sx_ReqInProgress390 THEN
	                #si_340DestinationA := 1;
	                #si_340DestinationB := 0;
	                #si_340DestinationC := 0;
	                #si_340DestinationD := 0;

	            ELSIF #iqUDT_WorkstationStatus."350".PEC_Eos.PEC THEN
	                #si_340DestinationA := 2;
	                #si_340DestinationB := 0;
	                #si_340DestinationC := 0;
	                #si_340DestinationD := 0;
	            ELSE
	                #si_340DestinationA := 0;
	                #si_340DestinationB := 0;
	                #si_340DestinationC := 0;
	                #si_340DestinationD := 0;
	            END_IF;


	            //Destinations from RAT 350
	            IF #sx_ActiveRequest380 AND NOT #sx_ReqInProgress380 THEN
	                #si_350DestinationA := 0;
	                #si_350DestinationB := 0;
	                #si_350DestinationC := 0;
	                #si_350DestinationD := 1;
	            ELSE
	                #si_350DestinationA := 0;
	                #si_350DestinationB := 0;
	                #si_350DestinationC := 0;
	                #si_350DestinationD := 0;
	            END_IF;

	            //Other destinations (stay the same as long as station is operating)
	            #si_240DestinationA := 1;
	            #si_240DestinationB := 0;
	            #si_240DestinationC := 0;
	            #si_240DestinationD := 1;

	            #si_360DestinationA := 1;
	            #si_360DestinationB := 2;
	            #si_360DestinationC := 0;
	            #si_360DestinationD := 0;

	            #si_370DestinationA := 1;
	            #si_370DestinationB := 2;
	            #si_370DestinationC := 2;
	            #si_370DestinationD := 0;
	        END_REGION
	        REGION Clear Right Station
	            //When clearing procedure is requested, set directions and destinations
	            IF NOT #ix_RightStationActive THEN

	                #sx_ClearRightStation := TRUE;

	                #sx_DirectionChange380 := TRUE;
	                #sx_DirectionChange390 := TRUE;

	                #si_340DestinationA := 1;
	                #si_340DestinationB := 0;
	                #si_340DestinationC := 0;
	                #si_340DestinationD := 0;

	                #si_350DestinationA := 0;
	                #si_350DestinationB := 0;
	                #si_350DestinationC := 0;
	                #si_350DestinationD := 1;

	                #si_360DestinationA := 2;
	                #si_360DestinationB := 2;
	                #si_360DestinationC := 0;
	                #si_360DestinationD := 0;

	                #si_370DestinationA := 2;
	                #si_370DestinationB := 2;
	                #si_370DestinationC := 2;
	                #si_370DestinationD := 0;
	            ELSE
	                #sx_ClearRightStation := FALSE;
	            END_IF;

	            //When clearing procedure is done reset directions
	            IF #s_F_Trig_ClearRight.Q THEN
	                #sx_DirectionChange380 := FALSE;
	                #sx_DirectionChange390 := FALSE;
	            END_IF;
	        END_REGION
	        REGION 310

	            REGION Displacement

	                #sFB_Displacement310(#sUDT_Interface_310);

	            END_REGION


	            REGION Conveyor
	                #sFB_Conveyor_310(iUDT_ConveyorConfiguration := #iUDT_Configuration."310".Conveyor,
	                                  idi_PECEoSDistance := 0,
	                                  idi_PECBoSDistance := 0,
	                                  ii_ExternalSpeed := 0,
	                                  ix_SafetyOk := #ix_SafetyOk,
	                                  ix_24vOk := #ix_24vOk,
	                                  ix_400vOk := #ix_400vOk,
	                                  ix_HardwareOk := #ix_HardwareOk,
	                                  ix_PECEoS := TRUE,
	                                  ix_PECBoS := TRUE,
	                                  ix_ExternalRequestHold := false,
	                                  qUDT_HMIStatus => #iqUDT_WorkstationStatus."310".Conveyor,
	                                  qUDT_Status => #iqUDT_WorkstationCommonStatus."310",
	                                  iqUDT_EquipmentControl := #iqUDT_EquipmentControl,
	                                  iqUDT_ConveyorCommand := #iqUDT_WorkstationCommands."310".Conveyor,
	                                  iqUDT_ConveyorInterface := #sUDT_Interface_310,
	                                  iqUDT_HandShakeUp := #iqUDT_HandshakeUpstream310,
	                                  iqUDT_HandShake := #sUDT_Handshake_310,
	                                  iqUDT_Statistics := #iqUDT_WorkstationStatistics."310".Conveyor);
	            END_REGION

	            REGION VFD

	                #sFB_VfdNORDPPO4_310(iUDT_VFDConfig := #iUDT_Configuration."310".VFD,
	                                     iUDT_VFDInputs := #iUDT_MotorInput310,
	                                     iUDT_MotorData := #iUDT_MotorData310,
	                                     ix_24vOk := #ix_24vOk,
	                                     ix_400vOk := #ix_400vOk,
	                                     ix_QuickStopDisable := TRUE,
	                                     ix_SimulationModeActive := "DB_Memory".Simulation,
	                                     qUDT_HMIStatus => #iqUDT_WorkstationStatus."310".VFD,
	                                     qUDT_VFDOutputs => #qUDT_MotorOutput310,
	                                     iqUDT_ConveyorInterface := #sUDT_Interface_310,
	                                     iqUDT_VFDStatistics := #iqUDT_WorkstationStatistics."310".VFD,
	                                     iqx_StartCommissioning := #iqx_StartComissioning310);

	            END_REGION
	        END_REGION


	        REGION 320

	            REGION Displacement

	                #sFB_Displacement320(#sUDT_Interface_320);

	            END_REGION

	            REGION Tracking

	                #sFB_Tracking_320(iUDT_ConveyorCommonConfiguration := #iUDT_Configuration."320".Conveyor.Common,
	                                  iqa_TrackingData := #sa_TrackingArray_320,
	                                  iqUDT_ConveyorInterface := #sUDT_Interface_320,
	                                  iqUDT_HandshakeUp := #sUDT_Handshake_310,
	                                  iqUDT_Handshake := #sUDT_Handshake_320);
	            END_REGION

	            REGION EOS

	                #sFB_PECUpdate_320(iUDT_PECUpdateConfiguration := #iUDT_Configuration."320".PEC_Eos,
	                                   iUDT_ConveyorCommonConfiguration := #iUDT_Configuration."320".Conveyor.Common,
	                                   ix_PEC := #iUDT_MotorInput320.AllSensorPortInputs.LeftSensor,
	                                   ix_TeachingMode := FALSE,
	                                   qUDT_Status => #iqUDT_WorkstationStatus."320".PEC_Eos,
	                                   qi_GINwrite => #ti_dummy,
	                                   qx_PECFiltered => #tx_dummy,
	                                   iqa_TrackingData := #sa_TrackingArray_320,
	                                   iqUDT_ConveyorInterface := #sUDT_Interface_320,
	                                   iqUDT_UnknownGINRange := #iqUDT_UnknownGINRange,
	                                   iqUDT_FifoHeader := "DB_FIFOLostGIN".Header,
	                                   iqa_FifoData := "DB_FIFOLostGIN".Data,
	                                   iqUDT_Statistics := #iqUDT_WorkstationStatistics."320".PEC_Eos);

	            END_REGION

	            REGION Conveyor
	                #sFB_Conveyor_320(iUDT_ConveyorConfiguration := #iUDT_Configuration."320".Conveyor,
	                                  idi_PECEoSDistance := #iUDT_Configuration."320".PEC_Eos.Distance,
	                                  idi_PECBoSDistance := 0,
	                                  ii_ExternalSpeed := 0,
	                                  ix_SafetyOk := #ix_SafetyOk,
	                                  ix_24vOk := #ix_24vOk,
	                                  ix_400vOk := #ix_400vOk,
	                                  ix_HardwareOk := #ix_HardwareOk,
	                                  ix_PECEoS := #iqUDT_WorkstationStatus."320".PEC_Eos.PEC,
	                                  ix_PECBoS := TRUE,
	                                  ix_ExternalRequestHold := FALSE,
	                                  qUDT_HMIStatus => #iqUDT_WorkstationStatus."320".Conveyor,
	                                  qUDT_Status => #iqUDT_WorkstationCommonStatus."320",
	                                  iqUDT_EquipmentControl := #iqUDT_EquipmentControl,
	                                  iqUDT_ConveyorCommand := #iqUDT_WorkstationCommands."320".Conveyor,
	                                  iqUDT_ConveyorInterface := #sUDT_Interface_320,
	                                  iqUDT_HandShakeUp := #sUDT_Handshake_310,
	                                  iqUDT_HandShake := #sUDT_Handshake_320,
	                                  iqUDT_Statistics := #iqUDT_WorkstationStatistics."320".Conveyor);
	            END_REGION

	            REGION MCO
	                #sFB_MCOConveyLinxAixController_320(iUDT_AixConfig := #iUDT_Configuration."320".MCO_M01,
	                                                    iUDT_AixInputsModule := #iUDT_MotorInput320,
	                                                    ix_24vOk := #ix_24vOk,
	                                                    ix_SimulationModeActive := "DB_Memory".Simulation,
	                                                    ii_MotorPositionId := 1,
	                                                    qUDT_HMIStatus => #iqUDT_WorkstationStatus."320".MCO_M01,
	                                                    iqUDT_AixOutputsModule := #qUDT_MotorOutput320,
	                                                    iqUDT_ConveyorInterface := #sUDT_Interface_320,
	                                                    iqUDT_MCOStatistics := #iqUDT_WorkstationStatistics."320".MCO_M01);
	            END_REGION


	        END_REGION
	        REGION 330

	            REGION Displacement

	                #sFB_Displacement330(#sUDT_Interface_330);

	            END_REGION

	            REGION Tracking

	                #sFB_Tracking_330(iUDT_ConveyorCommonConfiguration := #iUDT_Configuration."330".Conveyor.Common,
	                                  iqa_TrackingData := #sa_TrackingArray_330,
	                                  iqUDT_ConveyorInterface := #sUDT_Interface_330,
	                                  iqUDT_HandshakeUp := #sUDT_Handshake_320,
	                                  iqUDT_Handshake := #sUDT_Handshake_330);
	            END_REGION

	            REGION EOS

	                #sFB_PECUpdate_330(iUDT_PECUpdateConfiguration := #iUDT_Configuration."330".PEC_Eos,
	                                   iUDT_ConveyorCommonConfiguration := #iUDT_Configuration."330".Conveyor.Common,
	                                   ix_PEC := #iUDT_MotorInput320.AllSensorPortInputs.RightSensor,
	                                   ix_TeachingMode := FALSE,
	                                   qUDT_Status => #iqUDT_WorkstationStatus."330".PEC_Eos,
	                                   qi_GINwrite => #ti_dummy,
	                                   qx_PECFiltered => #tx_dummy,
	                                   iqa_TrackingData := #sa_TrackingArray_330,
	                                   iqUDT_ConveyorInterface := #sUDT_Interface_330,
	                                   iqUDT_UnknownGINRange := #iqUDT_UnknownGINRange,
	                                   iqUDT_FifoHeader := "DB_FIFOLostGIN".Header,
	                                   iqa_FifoData := "DB_FIFOLostGIN".Data,
	                                   iqUDT_Statistics := #iqUDT_WorkstationStatistics."330".PEC_Eos);

	            END_REGION

	            REGION Scanner

	                // #sFB_CognexDM260_330(iUDT_CognexDM260_IN    := #iUDT_ScannerInput330,
	                //                      qs_Barcode             => #ts_Barcode330,
	                //                      iqUDT_EquipmentControl := #iqUDT_EquipmentControl,
	                //                      ix_Trigger             := #sa_TrackingArray_330[50] > 0,
	                //                      qUDT_CognexDM260_OUT   => #qUDT_ScannerOutput330,
	                //                      qw_RetVal              => #tw_dummy);
	                //
	                //

	                // #sFB_Blade(iudt_DataLogicBladeIN := #iUDT_Blade_IN,
	                //            ix_Trigger            := #sa_TrackingArray_330[55] > 0,
	                //            qx_Trigger            => #qx_BladeOUT,
	                //            qs_Barcode            => #ts_Barcode330);
	                //
	                (*
	                #sFB_SickDemoo(ix_Trigger := #sa_TrackingArray_330[55] > 0 (*OR "DB_Test"."TRL03-141_Destination" = 2*),
	                               HWInputIdent := 714,
	                               HWInputLength := 32,
	                               HWOutputIdent := 716,
	                               HWOutputLength := 32,
	                               CANId := 0,
	                               qs_Barcode => #ts_Barcode330,
	                               iqUDT_EquipmentControl := #iqUDT_EquipmentControl);
	                *)
	                #iqUDT_ScannerInput330.Trigger := #sa_TrackingArray_330[55] > 0 (*OR "DB_Test"."TRL03-141_Destination" = 2*);
	                #ts_Barcode330 := #iqUDT_ScannerInput330.BarCodeValue;




	            END_REGION

	            REGION Conveyor
	                #sUDT_Handshake_330.RTR := #sUDT_Handshake_330.RTR OR #iqUDT_WorkstationStatus."330".PEC_Eos.PEC;
	                // #sx_Enable330 := #iUDT_MotorInput320.AllSensorPortInputs.RightSensor OR #iUDT_MotorInput390.AllSensorPortInputs.LeftSensor OR #iUDT_MotorInput350.AllSensorPortInputs.LeftSensor;
	                #sFB_Conveyor_330(iUDT_ConveyorConfiguration := #iUDT_Configuration."330".Conveyor,
	                                  idi_PECEoSDistance := #iUDT_Configuration."330".PEC_Eos.Distance,
	                                  idi_PECBoSDistance := 0,
	                                  ii_ExternalSpeed := 0,
	                                  ix_SafetyOk := #ix_SafetyOk,
	                                  ix_24vOk := #ix_24vOk,
	                                  ix_400vOk := #ix_400vOk,
	                                  ix_HardwareOk := #ix_HardwareOk,
	                                  ix_PECEoS := #iqUDT_WorkstationStatus."330".PEC_Eos.PEC,
	                                  ix_PECBoS := TRUE,
	                                  ix_ExternalRequestHold := false,
	                                  qUDT_HMIStatus => #iqUDT_WorkstationStatus."330".Conveyor,
	                                  qUDT_Status => #iqUDT_WorkstationCommonStatus."330",
	                                  iqUDT_EquipmentControl := #iqUDT_EquipmentControl,
	                                  iqUDT_ConveyorCommand := #iqUDT_WorkstationCommands."330".Conveyor,
	                                  iqUDT_ConveyorInterface := #sUDT_Interface_330,
	                                  iqUDT_HandShakeUp := #sUDT_Handshake_320,
	                                  iqUDT_HandShake := #sUDT_Handshake_330,
	                                  iqUDT_Statistics := #iqUDT_WorkstationStatistics."330".Conveyor);
	            END_REGION

	            REGION MCO
	                #sFB_MCOConveyLinxAixController_330(iUDT_AixConfig := #iUDT_Configuration."330".MCO_M01,
	                                                    iUDT_AixInputsModule := #iUDT_MotorInput320,
	                                                    ix_24vOk := #ix_24vOk,
	                                                    ix_SimulationModeActive := "DB_Memory".Simulation,
	                                                    ii_MotorPositionId := 2,
	                                                    qUDT_HMIStatus => #iqUDT_WorkstationStatus."330".MCO_M01,
	                                                    iqUDT_AixOutputsModule := #qUDT_MotorOutput320,
	                                                    iqUDT_ConveyorInterface := #sUDT_Interface_330,
	                                                    iqUDT_MCOStatistics := #iqUDT_WorkstationStatistics."330".MCO_M01);
	            END_REGION


	        END_REGION

	        REGION 340

	            REGION Displacement

	                #sFB_Displacement340(#sUDT_Interface_340);

	            END_REGION

	            REGION MCO
	                #sFB_MCOConveyLinxAixController_340(iUDT_AixConfig := #iUDT_Configuration."340".MCO_M01,
	                                                    iUDT_AixInputsModule := #iUDT_MotorInput340,
	                                                    ii_PositionSetpoint := #iqUDT_RATPositioning340.Lower.EndPosition,
	                                                    ix_24vOk := #ix_24vOk,
	                                                    ix_SimulationModeActive := "DB_Memory".Simulation,
	                                                    ii_MotorPositionId := 1,
	                                                    ix_StartPositioning := #iqUDT_RATPositioning340.Lower.Start,
	                                                    ix_ResetPosition := #iqUDT_RATPositioning340.Lower.ResetPosition,
	                                                    qUDT_HMIStatus => #iqUDT_WorkstationStatus."340".MCO_M01,
	                                                    qx_Positioned => #iqUDT_RATPositioning340.Lower.Done,
	                                                    iqUDT_AixOutputsModule := #qUDT_MotorOutput340,
	                                                    iqUDT_ConveyorInterface := #sUDT_Interface_340,
	                                                    iqUDT_MCOStatistics := #iqUDT_WorkstationStatistics."340".MCO_M01);
	            END_REGION


	        END_REGION
	        REGION 341

	            REGION Displacement

	                #sFB_Displacement341(#sUDT_Interface_341);

	            END_REGION

	            REGION RAT

	                #sFB_RightAngledTransfer_341(iUDT_Configuration := #iUDT_Configuration."341".RightAngledTransfer,
	                                             iUDT_LowerConveyorConfiguration := #iUDT_Configuration."340".Conveyor,
	                                             iUDT_UpperConveyorConfiguration := #iUDT_Configuration."341".Conveyor,
	                                             iUDT_PECConfiguration := #iUDT_Configuration."340".PEC_Eos,
	                                             ii_DestinationA := #si_340DestinationA,
	                                             ii_DestinationB := #si_340DestinationB,
	                                             ii_DestinationC := #si_340DestinationC,
	                                             ii_DestinationD := #si_340DestinationD,
	                                             ix_HardwareOk := #ix_HardwareOk,
	                                             ix_400vOk := #ix_400vOk,
	                                             ix_24vOk := #ix_24vOk,
	                                             ix_SafetyOk := #ix_SafetyOk,
	                                             ix_AirPressureOk := #ix_AirPressureOk,
	                                             ix_SectionIsDown := #ix_SectionIsDown341,
	                                             ix_SectionIsUp := #ix_SectionIsUp341,
	                                             ix_ConveyorAAuto := #iqUDT_WorkstationCommonStatus."330".AutoON,
	                                             ix_ConveyorBAuto := #iqUDT_WorkstationCommonStatus."370".AutoON,
	                                             ix_ConveyorCAuto := #iqUDT_WorkstationCommonStatus."351".AutoON,
	                                             ix_ConveyorDAuto := FALSE,
	                                             ix_PEC := #iUDT_MotorInput340.AllSensorPortInputs.LeftSensor,
	                                             ix_ExternalReceiveRequestA := NOT #iqUDT_WorkstationStatus."330".PEC_Eos.PEC,
	                                             ix_ExternalReceiveRequestB := false,
	                                             ix_ExternalReceiveRequestC := false,
	                                             ix_ExternalReceiveRequestD := false,
	                                             ix_PECInfeedA := #iqUDT_WorkstationStatus."330".PEC_Eos.PEC,
	                                             ix_PECInfeedB := #iqUDT_WorkstationStatus."370".PEC_Eos.PEC,
	                                             ix_PECInfeedC := #iqUDT_WorkstationStatus."350".PEC_Eos.PEC,
	                                             qUDT_HMIRATStatus => #iqUDT_WorkstationStatus."341".RightAngledTransfer,
	                                             qUDT_HMIConveyorStatus => #iqUDT_WorkstationStatus."340".Conveyor,
	                                             qUDT_HMIPECStatus => #iqUDT_WorkstationStatus."340".PEC_Eos,
	                                             qUDT_RATStatus => #iqUDT_WorkstationCommonStatus."341",
	                                             qUDT_ConveyorStatus => #iqUDT_WorkstationCommonStatus."340",
	                                             qx_PopupControl => #qx_PopupControl341,
	                                             iqUDT_EquipmentControl := #iqUDT_EquipmentControl,
	                                             iqUDT_RATCommand := #iqUDT_WorkstationCommands."341".RightAngledTransfer,
	                                             iqUDT_ConveyorCommand := #iqUDT_WorkstationCommands."340".Conveyor,
	                                             iqUDT_RATStatistics := #iqUDT_WorkstationStatistics."341".RightAngledTransfer,
	                                             iqUDT_ConveyorStatistics := #iqUDT_WorkstationStatistics."340".Conveyor,
	                                             iqUDT_PECStatistics := #iqUDT_WorkstationStatistics."340".PEC_Eos,
	                                             iqUDT_HandShakeConveyorA := #sUDT_Handshake_330,
	                                             iqUDT_HandShakeConveyorB := #sUDT_Handshake_340,
	                                             iqUDT_HandShakeConveyorC := #sUDT_HandshakeUp_341,
	                                             iqUDT_HandShakeConveyorD := #sUDT_Handshake_341,
	                                             iqUDT_LowerConveyorInterface := #sUDT_Interface_340,
	                                             iqUDT_UpperConveyorInterface := #sUDT_Interface_341,
	                                             iqUDT_RATPositioning := #iqUDT_RATPositioning340,
	                                             iqUDT_BladeStopEoSInterface := #tUDT_DummyBladeStop,
	                                             iqUDT_BladeStopBoSInterface := #tUDT_DummyBladeStop);

	            END_REGION

	            REGION MCO
	                #sFB_MCOConveyLinxAixController_341(iUDT_AixConfig := #iUDT_Configuration."341".MCO_M01,
	                                                    iUDT_AixInputsModule := #iUDT_MotorInput340,
	                                                    ix_24vOk := #ix_24vOk,
	                                                    ix_SimulationModeActive := "DB_Memory".Simulation,
	                                                    ii_MotorPositionId := 2,
	                                                    qUDT_HMIStatus => #iqUDT_WorkstationStatus."341".MCO_M01,
	                                                    iqUDT_AixOutputsModule := #qUDT_MotorOutput340,
	                                                    iqUDT_ConveyorInterface := #sUDT_Interface_341,
	                                                    iqUDT_MCOStatistics := #iqUDT_WorkstationStatistics."341".MCO_M01);
	            END_REGION

	        END_REGION

	        REGION 350

	            REGION Displacement

	                #sFB_Displacement350(#sUDT_Interface_350);

	            END_REGION

	            REGION MCO
	                #sFB_MCOConveyLinxAixController_350(iUDT_AixConfig := #iUDT_Configuration."350".MCO_M01,
	                                                    iUDT_AixInputsModule := #iUDT_MotorInput350,
	                                                    ix_24vOk := #ix_24vOk,
	                                                    ix_SimulationModeActive := "DB_Memory".Simulation,
	                                                    ii_MotorPositionId := 1,
	                                                    qUDT_HMIStatus => #iqUDT_WorkstationStatus."350".MCO_M01,
	                                                    iqUDT_AixOutputsModule := #qUDT_MotorOutput350,
	                                                    iqUDT_ConveyorInterface := #sUDT_Interface_350,
	                                                    iqUDT_MCOStatistics := #iqUDT_WorkstationStatistics."350".MCO_M01);
	            END_REGION

	        END_REGION

	        REGION 351

	            REGION Displacement

	                #sFB_Displacement351(#sUDT_Interface_351);

	            END_REGION

	            REGION RAT

	                #sFB_RightAngledTransfer_351(iUDT_Configuration := #iUDT_Configuration."351".RightAngledTransfer,
	                                             iUDT_LowerConveyorConfiguration := #iUDT_Configuration."350".Conveyor,
	                                             iUDT_UpperConveyorConfiguration := #iUDT_Configuration."351".Conveyor,
	                                             iUDT_PECConfiguration := #iUDT_Configuration."350".PEC_Eos,
	                                             ii_DestinationA := #si_350DestinationA,
	                                             ii_DestinationB := #si_350DestinationB,
	                                             ii_DestinationC := #si_350DestinationC,
	                                             ii_DestinationD := #si_350DestinationD,
	                                             ix_HardwareOk := #ix_HardwareOk,
	                                             ix_400vOk := #ix_400vOk,
	                                             ix_24vOk := #ix_24vOk,
	                                             ix_SafetyOk := #ix_SafetyOk,
	                                             ix_AirPressureOk := #ix_AirPressureOk,
	                                             ix_SectionIsDown := #ix_SectionIsDown351,
	                                             ix_SectionIsUp := #ix_SectionIsUp351,
	                                             ix_ConveyorAAuto := false,
	                                             ix_ConveyorBAuto := #iqUDT_WorkstationCommonStatus."360".AutoON,
	                                             ix_ConveyorCAuto := false,
	                                             ix_ConveyorDAuto := #iqUDT_WorkstationCommonStatus."341".AutoON,
	                                             ix_PEC := #iUDT_MotorInput350.AllSensorPortInputs.LeftSensor,
	                                             ix_ExternalReceiveRequestA := false,
	                                             ix_ExternalReceiveRequestB := false,
	                                             ix_ExternalReceiveRequestC := false,
	                                             ix_ExternalReceiveRequestD := #sFB_RightAngledTransfer_341.qx_ExternalSendRequestC,//NOT #iUDT_MotorInput340.AllSensorPortInputs.LeftSensor AND NOT #sx_ActiveRequest390,,,,,,,,
	                                             ix_PECInfeedB := #iqUDT_WorkstationStatus."360".PEC_Eos.PEC,
	                                             ix_PECInfeedD := #iqUDT_WorkstationStatus."340".PEC_Eos.PEC,
	                                             qUDT_HMIRATStatus => #iqUDT_WorkstationStatus."351".RightAngledTransfer,
	                                             qUDT_HMIConveyorStatus => #iqUDT_WorkstationStatus."350".Conveyor,
	                                             qUDT_HMIPECStatus => #iqUDT_WorkstationStatus."350".PEC_Eos,
	                                             qUDT_RATStatus => #iqUDT_WorkstationCommonStatus."351",
	                                             qUDT_ConveyorStatus => #iqUDT_WorkstationCommonStatus."350",
	                                             qx_PopupControl => #qx_PopupControl351,
	                                             iqUDT_EquipmentControl := #iqUDT_EquipmentControl,
	                                             iqUDT_RATCommand := #iqUDT_WorkstationCommands."351".RightAngledTransfer,
	                                             iqUDT_ConveyorCommand := #iqUDT_WorkstationCommands."350".Conveyor,
	                                             iqUDT_RATStatistics := #iqUDT_WorkstationStatistics."351".RightAngledTransfer,
	                                             iqUDT_ConveyorStatistics := #iqUDT_WorkstationStatistics."350".Conveyor,
	                                             iqUDT_PECStatistics := #iqUDT_WorkstationStatistics."350".PEC_Eos,
	                                             iqUDT_HandShakeConveyorA := #tUDT_dummyHandshake,
	                                             iqUDT_HandShakeConveyorB := #sUDT_Handshake_350,
	                                             iqUDT_HandShakeConveyorC := #tUDT_dummyHandshake,
	                                             iqUDT_HandShakeConveyorD := #sUDT_HandshakeUp_341,
	                                             iqUDT_LowerConveyorInterface := #sUDT_Interface_350,
	                                             iqUDT_UpperConveyorInterface := #sUDT_Interface_351,
	                                             iqUDT_RATPositioning := #iqUDT_RATPositioning350,
	                                             iqUDT_BladeStopEoSInterface := #tUDT_DummyBladeStop,
	                                             iqUDT_BladeStopBoSInterface := #tUDT_DummyBladeStop);

	            END_REGION

	            REGION MCO
	                #sFB_MCOConveyLinxAixController_351(iUDT_AixConfig := #iUDT_Configuration."351".MCO_M01,
	                                                    iUDT_AixInputsModule := #iUDT_MotorInput350,
	                                                    ii_PositionSetpoint := #iqUDT_RATPositioning350.Upper.EndPosition,
	                                                    ix_24vOk := #ix_24vOk,
	                                                    ix_SimulationModeActive := "DB_Memory".Simulation,
	                                                    ii_MotorPositionId := 2,
	                                                    ix_StartPositioning := #iqUDT_RATPositioning350.Upper.Start,
	                                                    ix_ResetPosition := #iqUDT_RATPositioning350.Upper.ResetPosition,
	                                                    qUDT_HMIStatus => #iqUDT_WorkstationStatus."351".MCO_M01,
	                                                    qx_Positioned => #iqUDT_RATPositioning350.Upper.Done,
	                                                    iqUDT_AixOutputsModule := #qUDT_MotorOutput350,
	                                                    iqUDT_ConveyorInterface := #sUDT_Interface_351,
	                                                    iqUDT_MCOStatistics := #iqUDT_WorkstationStatistics."351".MCO_M01);
	            END_REGION
	        END_REGION

	        REGION 360

	            REGION Displacement

	                #sFB_Displacement360(#sUDT_Interface_360);

	            END_REGION

	            REGION MCO
	                #sFB_MCOConveyLinxAixController_360(iUDT_AixConfig := #iUDT_Configuration."360".MCO_M01,
	                                                    iUDT_AixInputsModule := #iUDT_MotorInput360,
	                                                    ii_PositionSetpoint := #iqUDT_RATPositioning360.Lower.EndPosition,
	                                                    ix_24vOk := #ix_24vOk,
	                                                    ix_SimulationModeActive := "DB_Memory".Simulation,
	                                                    ii_MotorPositionId := 1,
	                                                    ix_StartPositioning := #iqUDT_RATPositioning360.Lower.Start,
	                                                    ix_ResetPosition := #iqUDT_RATPositioning360.Lower.ResetPosition,
	                                                    qUDT_HMIStatus => #iqUDT_WorkstationStatus."360".MCO_M01,
	                                                    qx_Positioned => #iqUDT_RATPositioning360.Lower.Done,
	                                                    iqUDT_AixOutputsModule := #qUDT_MotorOutput360,
	                                                    iqUDT_ConveyorInterface := #sUDT_Interface_360,
	                                                    iqUDT_MCOStatistics := #iqUDT_WorkstationStatistics."360".MCO_M01);
	            END_REGION

	        END_REGION
	        REGION 361

	            REGION Displacement

	                #sFB_Displacement361(#sUDT_Interface_361);

	            END_REGION

	            REGION RAT

	                #sFB_RightAngledTransfer_361(iUDT_Configuration := #iUDT_Configuration."361".RightAngledTransfer,
	                                             iUDT_LowerConveyorConfiguration := #iUDT_Configuration."360".Conveyor,
	                                             iUDT_UpperConveyorConfiguration := #iUDT_Configuration."361".Conveyor,
	                                             iUDT_PECConfiguration := #iUDT_Configuration."360".PEC_Eos,
	                                             ii_DestinationA := #si_360DestinationA,
	                                             ii_DestinationB := #si_360DestinationB,
	                                             ii_DestinationC := #si_360DestinationC,
	                                             ii_DestinationD := #si_360DestinationD,
	                                             ix_HardwareOk := #ix_HardwareOk,
	                                             ix_400vOk := #ix_400vOk,
	                                             ix_24vOk := #ix_24vOk,
	                                             ix_SafetyOk := #ix_SafetyOk,
	                                             ix_AirPressureOk := #ix_AirPressureOk,
	                                             ix_SectionIsDown := #ix_SectionIsDown361,
	                                             ix_SectionIsUp := #ix_SectionIsUp361,
	                                             ix_ConveyorAAuto := #iqUDT_WorkstationCommonStatus."350".AutoON,
	                                             ix_ConveyorBAuto := #iqUDT_WorkstationCommonStatus."380".AutoON,
	                                             ix_ConveyorCAuto := FALSE,
	                                             ix_ConveyorDAuto := #iqUDT_WorkstationCommonStatus."371".AutoON,
	                                             ix_PEC := #iUDT_MotorInput360.AllSensorPortInputs.LeftSensor,
	                                             ix_ExternalReceiveRequestA := #sFB_RightAngledTransfer_351.qx_ExternalSendRequestB AND (#sx_ActiveRequest380 OR #sx_ClearRightStation),//#sx_ActiveRequest380 AND NOT #iUDT_MotorInput350.AllSensorPortInputs.LeftSensor,
	                                             ix_ExternalReceiveRequestB := (#sx_TransferOut380 OR #sx_ClearRightStation) AND NOT #iqUDT_WorkstationStatus."380".PEC_Eos.PEC,
	                                             ix_ExternalReceiveRequestC := false,
	                                             ix_ExternalReceiveRequestD := false,
	                                             ix_PECInfeedA := #iqUDT_WorkstationStatus."350".PEC_Eos.PEC,
	                                             ix_PECInfeedB := #iqUDT_WorkstationStatus."380".PEC_Eos.PEC,
	                                             ix_PECInfeedD := #iqUDT_WorkstationStatus."370".PEC_Eos.PEC,
	                                             qUDT_HMIRATStatus => #iqUDT_WorkstationStatus."361".RightAngledTransfer,
	                                             qUDT_HMIConveyorStatus => #iqUDT_WorkstationStatus."360".Conveyor,
	                                             qUDT_HMIPECStatus => #iqUDT_WorkstationStatus."360".PEC_Eos,
	                                             qUDT_RATStatus => #iqUDT_WorkstationCommonStatus."361",
	                                             qUDT_ConveyorStatus => #iqUDT_WorkstationCommonStatus."360",
	                                             qx_PopupControl => #qx_PopupControl361,
	                                             iqUDT_EquipmentControl := #iqUDT_EquipmentControl,
	                                             iqUDT_RATCommand := #iqUDT_WorkstationCommands."361".RightAngledTransfer,
	                                             iqUDT_ConveyorCommand := #iqUDT_WorkstationCommands."360".Conveyor,
	                                             iqUDT_RATStatistics := #iqUDT_WorkstationStatistics."361".RightAngledTransfer,
	                                             iqUDT_ConveyorStatistics := #iqUDT_WorkstationStatistics."360".Conveyor,
	                                             iqUDT_PECStatistics := #iqUDT_WorkstationStatistics."360".PEC_Eos,
	                                             iqUDT_HandShakeConveyorA := #sUDT_Handshake_350,
	                                             iqUDT_HandShakeConveyorB := #sUDT_Handshake_360,
	                                             iqUDT_HandShakeConveyorC := #tUDT_dummyHandshake,
	                                             iqUDT_HandShakeConveyorD := #sUDT_Handshake_361,
	                                             iqUDT_LowerConveyorInterface := #sUDT_Interface_360,
	                                             iqUDT_UpperConveyorInterface := #sUDT_Interface_361,
	                                             iqUDT_RATPositioning := #iqUDT_RATPositioning360,
	                                             iqUDT_BladeStopEoSInterface := #tUDT_DummyBladeStop,
	                                             iqUDT_BladeStopBoSInterface := #tUDT_DummyBladeStop);

	            END_REGION

	            REGION MCO
	                #sFB_MCOConveyLinxAixController_361(iUDT_AixConfig := #iUDT_Configuration."361".MCO_M01,
	                                                    iUDT_AixInputsModule := #iUDT_MotorInput360,
	                                                    ix_24vOk := #ix_24vOk,
	                                                    ix_SimulationModeActive := "DB_Memory".Simulation,
	                                                    ii_MotorPositionId := 2,
	                                                    qUDT_HMIStatus => #iqUDT_WorkstationStatus."361".MCO_M01,
	                                                    iqUDT_AixOutputsModule := #qUDT_MotorOutput360,
	                                                    iqUDT_ConveyorInterface := #sUDT_Interface_361,
	                                                    iqUDT_MCOStatistics := #iqUDT_WorkstationStatistics."361".MCO_M01);
	            END_REGION

	        END_REGION

	        REGION 370

	            REGION Displacement

	                #sFB_Displacement370(#sUDT_Interface_370);

	            END_REGION

	            REGION MCO
	                #sFB_MCOConveyLinxAixController_370(iUDT_AixConfig := #iUDT_Configuration."370".MCO_M01,
	                                                    iUDT_AixInputsModule := #iUDT_MotorInput370,
	                                                    ii_PositionSetpoint := #iqUDT_RATPositioning370.Lower.EndPosition,
	                                                    ix_24vOk := #ix_24vOk,
	                                                    ix_SimulationModeActive := "DB_Memory".Simulation,
	                                                    ii_MotorPositionId := 1,
	                                                    ix_StartPositioning := #iqUDT_RATPositioning370.Lower.Start,
	                                                    ix_ResetPosition := #iqUDT_RATPositioning370.Lower.ResetPosition,
	                                                    qUDT_HMIStatus => #iqUDT_WorkstationStatus."370".MCO_M01,
	                                                    qx_Positioned => #iqUDT_RATPositioning370.Lower.Done,
	                                                    iqUDT_AixOutputsModule := #qUDT_MotorOutput370,
	                                                    iqUDT_ConveyorInterface := #sUDT_Interface_370,
	                                                    iqUDT_MCOStatistics := #iqUDT_WorkstationStatistics."370".MCO_M01);
	            END_REGION


	        END_REGION
	        REGION 371

	            REGION Displacement

	                #sFB_Displacement371(#sUDT_Interface_371);

	            END_REGION

	            REGION RAT

	                #sFB_RightAngledTransfer_371(iUDT_Configuration := #iUDT_Configuration."371".RightAngledTransfer,
	                                             iUDT_LowerConveyorConfiguration := #iUDT_Configuration."370".Conveyor,
	                                             iUDT_UpperConveyorConfiguration := #iUDT_Configuration."371".Conveyor,
	                                             iUDT_PECConfiguration := #iUDT_Configuration."370".PEC_Eos,
	                                             ii_DestinationA := #si_370DestinationA,
	                                             ii_DestinationB := #si_370DestinationB,
	                                             ii_DestinationC := #si_370DestinationC,
	                                             ii_DestinationD := #si_370DestinationD,
	                                             ix_HardwareOk := #ix_HardwareOk,
	                                             ix_400vOk := #ix_400vOk,
	                                             ix_24vOk := #ix_24vOk,
	                                             ix_SafetyOk := #ix_SafetyOk,
	                                             ix_AirPressureOk := #ix_AirPressureOk,
	                                             ix_SectionIsDown := #ix_SectionIsDown371,
	                                             ix_SectionIsUp := #ix_SectionIsUp371,
	                                             ix_ConveyorAAuto := #iqUDT_WorkstationCommonStatus."340".AutoON,
	                                             ix_ConveyorBAuto := #iqUDT_WorkstationCommonStatus."390".AutoON,
	                                             ix_ConveyorCAuto := #iqUDT_WorkstationCommonStatus."361".AutoON,
	                                             ix_ConveyorDAuto := #iqUDT_WorkstationCommonStatus."241".AutoON,
	                                             ix_PEC := #iUDT_MotorInput370.AllSensorPortInputs.LeftSensor,
	                                             ix_ExternalReceiveRequestA := #sFB_RightAngledTransfer_341.qx_ExternalSendRequestB,
	                                             ix_ExternalReceiveRequestB := (#sx_TransferOut390 OR #sx_ClearRightStation) AND NOT #iqUDT_WorkstationStatus."390".PEC_Eos.PEC,
	                                             ix_ExternalReceiveRequestC := #sFB_RightAngledTransfer_361.qx_ExternalSendRequestD,
	                                             ix_ExternalReceiveRequestD := false,
	                                             ix_PECInfeedA := #iqUDT_WorkstationStatus."340".PEC_Eos.PEC,
	                                             ix_PECInfeedB := #iqUDT_WorkstationStatus."390".PEC_Eos.PEC,
	                                             ix_PECInfeedC := #iqUDT_WorkstationStatus."360".PEC_Eos.PEC,
	                                             ix_PECInfeedD := #iqUDT_WorkstationStatus."240".PEC_Eos.PEC,
	                                             qUDT_HMIRATStatus => #iqUDT_WorkstationStatus."371".RightAngledTransfer,
	                                             qUDT_HMIConveyorStatus => #iqUDT_WorkstationStatus."370".Conveyor,
	                                             qUDT_HMIPECStatus => #iqUDT_WorkstationStatus."370".PEC_Eos,
	                                             qUDT_RATStatus => #iqUDT_WorkstationCommonStatus."371",
	                                             qUDT_ConveyorStatus => #iqUDT_WorkstationCommonStatus."370",
	                                             qx_PopupControl => #qx_PopupControl371,
	                                             iqUDT_EquipmentControl := #iqUDT_EquipmentControl,
	                                             iqUDT_RATCommand := #iqUDT_WorkstationCommands."371".RightAngledTransfer,
	                                             iqUDT_ConveyorCommand := #iqUDT_WorkstationCommands."370".Conveyor,
	                                             iqUDT_RATStatistics := #iqUDT_WorkstationStatistics."371".RightAngledTransfer,
	                                             iqUDT_ConveyorStatistics := #iqUDT_WorkstationStatistics."370".Conveyor,
	                                             iqUDT_PECStatistics := #iqUDT_WorkstationStatistics."370".PEC_Eos,
	                                             iqUDT_HandShakeConveyorA := #sUDT_Handshake_340,
	                                             iqUDT_HandShakeConveyorB := #sUDT_Handshake_370,
	                                             iqUDT_HandShakeConveyorC := #sUDT_Handshake_361,
	                                             iqUDT_HandShakeConveyorD := #sUDT_Handshake_371,
	                                             iqUDT_LowerConveyorInterface := #sUDT_Interface_370,
	                                             iqUDT_UpperConveyorInterface := #sUDT_Interface_371,
	                                             iqUDT_RATPositioning := #iqUDT_RATPositioning370,
	                                             iqUDT_BladeStopEoSInterface := #tUDT_DummyBladeStop,
	                                             iqUDT_BladeStopBoSInterface := #tUDT_DummyBladeStop);

	            END_REGION

	            REGION MCO
	                #sFB_MCOConveyLinxAixController_371(iUDT_AixConfig := #iUDT_Configuration."371".MCO_M01,
	                                                    iUDT_AixInputsModule := #iUDT_MotorInput370,
	                                                    ii_PositionSetpoint := #iqUDT_RATPositioning370.Upper.EndPosition,
	                                                    ix_24vOk := #ix_24vOk,
	                                                    ix_SimulationModeActive := "DB_Memory".Simulation,
	                                                    ii_MotorPositionId := 2,
	                                                    ix_StartPositioning := #iqUDT_RATPositioning370.Upper.Start,
	                                                    ix_ResetPosition := #iqUDT_RATPositioning370.Upper.ResetPosition,
	                                                    qUDT_HMIStatus => #iqUDT_WorkstationStatus."371".MCO_M01,
	                                                    qx_Positioned => #iqUDT_RATPositioning370.Upper.Done,
	                                                    iqUDT_AixOutputsModule := #qUDT_MotorOutput370,
	                                                    iqUDT_ConveyorInterface := #sUDT_Interface_371,
	                                                    iqUDT_MCOStatistics := #iqUDT_WorkstationStatistics."371".MCO_M01);
	            END_REGION
	        END_REGION

	        REGION 380

	            REGION Displacement

	                #sFB_Displacement380(#sUDT_Interface_380);

	            END_REGION

	            REGION Tracking

	                #sFB_Tracking_380(iUDT_ConveyorCommonConfiguration := #iUDT_Configuration."380".Conveyor.Common,
	                                  iqa_TrackingData := #sa_TrackingArray_380,
	                                  iqUDT_ConveyorInterface := #sUDT_Interface_380,
	                                  iqUDT_HandshakeUp := #sUDT_Handshake_360,
	                                  iqUDT_Handshake := #sUDT_Handshake_380);
	            END_REGION

	            REGION EOS

